    // EN: Fallback after override release.
    //     The discharge sequence should normally keep override active
    //     during return. If override is released unexpectedly, return to
    //     programmed position automatically.
    backstopLatchedTargetPositionMm := backstopProgrammedTargetPositionMm;
    backstopPositioningRequestActive := TRUE;

END_IF;


//==============================================================
// 5.2) Active target selection
//==============================================================
// EN: Discharge override has priority even if normal automatic mode is off.
//     Without override or positioning request, target remains latched,
//     but the axis does not move.
// PT: Override de descarte tem prioridade mesmo com o automático normal desligado.
IF systemRunEnable AND backstopTargetOverrideActive THEN

    backstopTargetPositionMm :=
        LIMIT(
            machineConfig.backstopMinPositionMm,
            backstopTargetOverridePositionMm,
            machineConfig.backstopMaxPositionMm
        );

ELSE

    backstopTargetPositionMm :=
        LIMIT(
            machineConfig.backstopMinPositionMm,
            backstopLatchedTargetPositionMm,
            machineConfig.backstopMaxPositionMm
        );

END_IF;


//==============================================================
// 5.4) Home running flag
//==============================================================
IF (backstopControlState = 10) OR
   (backstopControlState = 11) OR
   (backstopControlState = 12) OR
   (backstopControlState = 13) OR
   (backstopControlState = 14) THEN

    backstopHomeRunning := TRUE;

ELSE

    backstopHomeRunning := FALSE;

END_IF;


//==============================================================
// 6) Position error calculation
//==============================================================
backstopPositionErrorMm :=
    backstopTargetPositionMm - backstopPositionMm;

backstopAbsPositionErrorMm :=
    ABS(backstopPositionErrorMm);

backstopInPosition :=
    backstopHomed AND
    (backstopAbsPositionErrorMm <= machineConfig.backstopPositionToleranceMm);


//==============================================================
// 7) Reset fault command
//==============================================================
IF resetCmd THEN

    IF safetyCircuitOk AND
       backstopDriveOk AND
       NOT backstopSafeMaxLimit AND
       NOT backstopSafeMinLimit THEN

        backstopFault := FALSE;
        backstopFaultCode := 0;

        IF backstopControlState = 40 THEN
            backstopControlState := 0;
        END_IF

    END_IF

END_IF;


//==============================================================
// 8) General protection
//==============================================================
IF NOT safetyCircuitOk THEN

    backstopState := 'SAFETY_OFF';

    tonBackstopHomingTimeout(IN := FALSE);
    tonBackstopHomeSettleDelay(IN := FALSE);

    backstopFault := TRUE;
    backstopFaultCode := 2;
    backstopControlState := 40;


ELSIF NOT backstopDriveOk THEN

    backstopState := 'DRIVE_NOT_OK';

    tonBackstopHomingTimeout(IN := FALSE);
    tonBackstopHomeSettleDelay(IN := FALSE);

    backstopFault := TRUE;
    backstopFaultCode := 1;
    backstopControlState := 40;


ELSIF backstopSafeMaxLimit THEN

    backstopState := 'SAFE_MAX_LIMIT';

    tonBackstopHomingTimeout(IN := FALSE);
    tonBackstopHomeSettleDelay(IN := FALSE);

    backstopFault := TRUE;
    backstopFaultCode := 6;
    backstopControlState := 40;


ELSIF backstopSafeMinLimit THEN

    backstopState := 'SAFE_MIN_LIMIT';

    tonBackstopHomingTimeout(IN := FALSE);
    tonBackstopHomeSettleDelay(IN := FALSE);

    backstopFault := TRUE;
    backstopFaultCode := 7;
    backstopControlState := 40;


ELSIF machineConfig.backstopHomeDirection = 0 THEN

    backstopState := 'INVALID_HOME_DIR';

    tonBackstopHomingTimeout(IN := FALSE);
    tonBackstopHomeSettleDelay(IN := FALSE);

    backstopFault := TRUE;
    backstopFaultCode := 5;
    backstopControlState := 40;


ELSIF NOT systemRunEnable THEN

    // EN: Master stop disables movement without generating an axis fault.
    backstopState := 'SYSTEM_DISABLED';

    backstopSignedSpeedRefMmps := 0.0;

    tonBackstopHomingTimeout(IN := FALSE);
    tonBackstopHomeSettleDelay(IN := FALSE);

    backstopPositioningRequestActive := FALSE;

    IF backstopControlState <> 40 THEN
        backstopControlState := 0;
    END_IF


ELSE

    //==============================================================
    // 9) Mode selection
    //==============================================================
    // EN: Homing has priority over manual and automatic positioning.
    IF rBackstopHome AND NOT backstopFault THEN
        backstopControlState := 10;
    END_IF;


    //==============================================================
    // 10) Backstop state machine
    //==============================================================
    CASE backstopControlState OF

        0: // STOP
            backstopState := 'STOP';

            tonBackstopHomingTimeout(IN := FALSE);
            tonBackstopHomeSettleDelay(IN := FALSE);

            // EN: Manual is allowed even with auto enabled,
            //     but not during automatic cycle override.
            IF (backstopOpenCmd OR backstopCloseCmd) AND
               NOT backstopTargetOverrideActive THEN

                backstopControlState := 20;


            ELSIF backstopTargetOverrideActive OR
                  (
                      backstopAutoCmd AND
                      backstopPositioningRequestActive
                  ) THEN

                backstopControlState := 30;

            END_IF


        10: // HOME_FAST_SEARCH
            backstopState := 'HOME_FAST';

            backstopHomed := FALSE;
            backstopInPosition := FALSE;

            tonBackstopHomeSettleDelay(IN := FALSE);

            tonBackstopHomingTimeout(
                IN := TRUE,
                PT := machineConfig.backstopHomingTimeout
            );

            IF tonBackstopHomingTimeout.Q THEN

                backstopSignedSpeedRefMmps := 0.0;

                tonBackstopHomingTimeout(IN := FALSE);

                backstopFault := TRUE;
                backstopFaultCode := 3;

                backstopState := 'HOME_TIMEOUT';
                backstopControlState := 40;


            ELSIF backstopHomeLimitReached THEN

                backstopSignedSpeedRefMmps := 0.0;

                backstopControlState := 11;


            ELSE

                IF backstopHomeMoveAllowed THEN

                    IF machineConfig.backstopHomeDirection > 0 THEN

                        backstopSignedSpeedRefMmps :=
                            ABS(machineConfig.backstopHomingSpeedMmps);

                    ELSE

                        backstopSignedSpeedRefMmps :=
                            -ABS(machineConfig.backstopHomingSpeedMmps);

                    END_IF

                ELSE

                    backstopSignedSpeedRefMmps := 0.0;

                END_IF

            END_IF


        11: // HOME_SLOW_EXIT_SENSOR
            backstopState := 'HOME_SLOW_EXIT';

            tonBackstopHomeSettleDelay(IN := FALSE);

            tonBackstopHomingTimeout(
                IN := TRUE,
                PT := machineConfig.backstopHomingTimeout
            );

            IF tonBackstopHomingTimeout.Q THEN

                backstopSignedSpeedRefMmps := 0.0;

                tonBackstopHomingTimeout(IN := FALSE);

                backstopFault := TRUE;
                backstopFaultCode := 3;

                backstopState := 'HOME_TIMEOUT';
                backstopControlState := 40;


            ELSIF backstopHomeLimitFallingEdge THEN

                backstopSignedSpeedRefMmps := 0.0;

                tonBackstopHomingTimeout(IN := FALSE);

                backstopControlState := 12;


            ELSE

                IF backstopHomeMoveAllowed THEN

                    IF machineConfig.backstopHomeDirection > 0 THEN

                        backstopSignedSpeedRefMmps :=
                            -ABS(machineConfig.backstopMinMoveSpeedMmps);

                    ELSE

                        backstopSignedSpeedRefMmps :=
                            ABS(machineConfig.backstopMinMoveSpeedMmps);

                    END_IF

                ELSE

                    backstopSignedSpeedRefMmps := 0.0;

                END_IF

            END_IF


        12: // HOME_SET_ENCODER
            backstopState := 'HOME_SET_ENCODER';

            backstopSignedSpeedRefMmps := 0.0;

            tonBackstopHomingTimeout(IN := FALSE);
            tonBackstopHomeSettleDelay(IN := FALSE);

            // EN: Set encoder to configured known home position.
            backstopSetEncoderPositionTrigger := TRUE;
            backstopSetEncoderPositionMm := machineConfig.backstopHomePositionMm;

            backstopHomed := TRUE;
            backstopFault := FALSE;
            backstopFaultCode := 0;

            // EN: After homing, latch current programmed target for home move.
            backstopLatchedTargetPositionMm := backstopProgrammedTargetPositionMm;
            backstopPositioningRequestActive := TRUE;

            // EN: Homing cancels previous manual intervention memory.
            backstopManualInterventionActive := FALSE;
            backstopManualInterventionPositionMm := 0.0;

            backstopControlState := 13;


        13: // HOME_WAIT_AFTER_SET
            backstopState := 'HOME_WAIT';

            backstopSignedSpeedRefMmps := 0.0;

            tonBackstopHomingTimeout(IN := FALSE);

            // EN: Fixed wait after encoder set.
            tonBackstopHomeSettleDelay(
                IN := TRUE,
                PT := T#5S
            );

            IF tonBackstopHomeSettleDelay.Q THEN

                tonBackstopHomeSettleDelay(IN := FALSE);

                backstopControlState := 14;

            END_IF


        14: // HOME_MOVE_TO_TARGET
            backstopState := 'HOME_TO_TARGET';

            tonBackstopHomingTimeout(IN := FALSE);
            tonBackstopHomeSettleDelay(IN := FALSE);

            // EN: Move to the latched programmed target after homing.
            IF backstopInPosition THEN

                backstopSignedSpeedRefMmps := 0.0;

                backstopPositioningRequestActive := FALSE;

                // EN: Home positioning completed, no manual intervention pending.
                backstopManualInterventionActive := FALSE;
                backstopManualInterventionPositionMm := 0.0;

                backstopControlState := 0;


            ELSE

                backstopRawSpeedRefMmps :=
                    backstopPositionErrorMm * machineConfig.backstopPositionKp;

                backstopRawSpeedRefMmps :=
                    LIMIT(
                        -ABS(machineConfig.backstopAutoMaxSpeedMmps),
                        backstopRawSpeedRefMmps,
                        ABS(machineConfig.backstopAutoMaxSpeedMmps)
                    );

                IF ABS(backstopRawSpeedRefMmps) <
                   ABS(machineConfig.backstopMinMoveSpeedMmps) THEN

                    IF backstopPositionErrorMm > 0.0 THEN

                        backstopRawSpeedRefMmps :=
                            ABS(machineConfig.backstopMinMoveSpeedMmps);

                    ELSE

                        backstopRawSpeedRefMmps :=
                            -ABS(machineConfig.backstopMinMoveSpeedMmps);

                    END_IF

                END_IF

                IF (backstopRawSpeedRefMmps > 0.0) AND backstopOpenAllowed THEN

                    backstopSignedSpeedRefMmps := backstopRawSpeedRefMmps;

                ELSIF (backstopRawSpeedRefMmps < 0.0) AND backstopCloseAllowed THEN

                    backstopSignedSpeedRefMmps := backstopRawSpeedRefMmps;

                ELSE

                    backstopSignedSpeedRefMmps := 0.0;

                END_IF

            END_IF


        20: // MANUAL
            backstopState := 'MANUAL';

            tonBackstopHomingTimeout(IN := FALSE);
            tonBackstopHomeSettleDelay(IN := FALSE);

            // EN: If automatic override starts, manual is cancelled.
            IF backstopTargetOverrideActive THEN

                backstopSignedSpeedRefMmps := 0.0;
                backstopControlState := 30;


            ELSIF backstopOpenCmd AND backstopCloseCmd THEN

                backstopSignedSpeedRefMmps := 0.0;


            ELSIF backstopOpenCmd THEN

                IF backstopOpenAllowed THEN

                    backstopSignedSpeedRefMmps :=
                        ABS(machineConfig.backstopManualSpeedMmps);

                    // EN: Store last manual intervention position.
                    //     This is updated while the operator holds the manual command.
                    backstopManualInterventionActive := TRUE;
                    backstopManualInterventionPositionMm := backstopPositionMm;

                ELSE

                    backstopSignedSpeedRefMmps := 0.0;

                END_IF


            ELSIF backstopCloseCmd THEN

                IF backstopCloseAllowed THEN

                    backstopSignedSpeedRefMmps :=
                        -ABS(machineConfig.backstopManualSpeedMmps);

                    // EN: Store last manual intervention position.
                    //     Even if operator closes, the discharge sequence will use
                    //     MAX(programmed position, manual position), so it remains safe.
                    backstopManualInterventionActive := TRUE;
                    backstopManualInterventionPositionMm := backstopPositionMm;

                ELSE

                    backstopSignedSpeedRefMmps := 0.0;

                END_IF


            ELSE

                backstopSignedSpeedRefMmps := 0.0;

                // EN: After manual command release, do not automatically return
                //     to programmed position. Wait for execute positioning command.
                backstopPositioningRequestActive := FALSE;

                backstopControlState := 0;

            END_IF


        30: // AUTO_POSITION
            backstopState := 'AUTO_POSITION';

            tonBackstopHomingTimeout(IN := FALSE);
            tonBackstopHomeSettleDelay(IN := FALSE);

            IF NOT backstopAutoCmd AND
               NOT backstopTargetOverrideActive THEN

                backstopSignedSpeedRefMmps := 0.0;
                backstopPositioningRequestActive := FALSE;
                backstopControlState := 0;


            ELSIF NOT backstopHomed THEN

                backstopSignedSpeedRefMmps := 0.0;
                backstopState := 'AUTO_NO_HOME';


            ELSIF (backstopOpenCmd OR backstopCloseCmd) AND
                  NOT backstopTargetOverrideActive THEN

                // EN: Manual has priority only outside automatic cycle override.
                backstopSignedSpeedRefMmps := 0.0;
                backstopPositioningRequestActive := FALSE;
                backstopControlState := 20;


            ELSIF NOT backstopTargetOverrideActive AND
                  NOT backstopPositioningRequestActive THEN

                // EN: Auto enabled but no positioning command active.
                backstopSignedSpeedRefMmps := 0.0;
                backstopControlState := 0;


            ELSIF backstopInPosition THEN

                backstopSignedSpeedRefMmps := 0.0;

                // EN: Normal positioning command ends when target is reached.
                //     Override remains controlled by the automatic cycle.
                IF NOT backstopTargetOverrideActive THEN

                    backstopPositioningRequestActive := FALSE;

                    // EN: If the backstop returned to programmed target,
                    //     clear previous manual intervention memory.
                    backstopManualInterventionActive := FALSE;
                    backstopManualInterventionPositionMm := 0.0;

                    backstopControlState := 0;

                END_IF


            ELSE

                backstopRawSpeedRefMmps :=
                    backstopPositionErrorMm * machineConfig.backstopPositionKp;

                backstopRawSpeedRefMmps :=
                    LIMIT(
                        -ABS(machineConfig.backstopAutoMaxSpeedMmps),
                        backstopRawSpeedRefMmps,
                        ABS(machineConfig.backstopAutoMaxSpeedMmps)
                    );

                IF ABS(backstopRawSpeedRefMmps) <
                   ABS(machineConfig.backstopMinMoveSpeedMmps) THEN

                    IF backstopPositionErrorMm > 0.0 THEN

                        backstopRawSpeedRefMmps :=
                            ABS(machineConfig.backstopMinMoveSpeedMmps);

                    ELSE

                        backstopRawSpeedRefMmps :=
                            -ABS(machineConfig.backstopMinMoveSpeedMmps);

                    END_IF

                END_IF

                IF (backstopRawSpeedRefMmps > 0.0) AND backstopOpenAllowed THEN

                    backstopSignedSpeedRefMmps := backstopRawSpeedRefMmps;

                ELSIF (backstopRawSpeedRefMmps < 0.0) AND backstopCloseAllowed THEN

                    backstopSignedSpeedRefMmps := backstopRawSpeedRefMmps;

                ELSE

                    backstopSignedSpeedRefMmps := 0.0;

                END_IF

            END_IF


        40: // FAULT
            backstopState := 'FAULT';

            backstopSignedSpeedRefMmps := 0.0;

            tonBackstopHomingTimeout(IN := FALSE);
            tonBackstopHomeSettleDelay(IN := FALSE);

            backstopPositioningRequestActive := FALSE;

            IF resetCmd AND
               safetyCircuitOk AND
               backstopDriveOk AND
               NOT backstopSafeMaxLimit AND
               NOT backstopSafeMinLimit THEN

                backstopFault := FALSE;
                backstopFaultCode := 0;
                backstopControlState := 0;

            END_IF


    ELSE

        backstopControlState := 0;

    END_CASE;

END_IF;


//==============================================================
// 11) Encoder set pulse
//==============================================================
// EN: Extend encoder set command to ensure the encoder block sees it.
tpBackstopSetEncoderPosition(
    IN := backstopSetEncoderPositionTrigger,
    PT := machineConfig.backstopSetEncoderPulseTime
);

backstopSetEncoderPosition := tpBackstopSetEncoderPosition.Q;


//==============================================================
// 12) Backstop drive direction and speed outputs
//==============================================================
// EN: Convert signed internal speed command into direction outputs
//     and positive speed reference.
IF systemRunEnable AND
   safetyCircuitOk AND
   backstopDriveOk AND
   NOT backstopFault AND
   (ABS(backstopSignedSpeedRefMmps) >= machineConfig.backstopRunMinSpeedMmps) THEN

    // EN: The servo receives the signed speed reference directly.
    // PT: O servo recebe diretamente a referência de velocidade com sinal.
    backstopSpeedRefMmps := backstopSignedSpeedRefMmps;

    backstopRunFw :=
        backstopSignedSpeedRefMmps > 0.0;

    backstopRunRev :=
        backstopSignedSpeedRefMmps < 0.0;

ELSE

    backstopSpeedRefMmps := 0.0;

    backstopRunFw := FALSE;
    backstopRunRev := FALSE;

END_IF;

// EN: Enable the servo with the stacker system; drive-ready feedback is not used here
//     because it would create a circular enable dependency.
// PT: Habilita o servo com o sistema do stacker; o retorno de drive pronto não é usado
//     aqui porque criaria uma dependência circular de habilitação.
backstopDriveEnable := systemRunEnable AND safetyCircuitOk;


//==============================================================
// 13) Backstop plate lift solenoid
//==============================================================
// EN: Lift the backstop plate during backstop movement and homing.
//     Discharge conveyor protection can be ORed after all methods are called.
IF systemRunEnable AND
   (
       backstopRunFw OR
       backstopRunRev OR
       sheetStackDischargeConveyorRun OR
       (backstopControlState = 10) OR
       (backstopControlState = 11) OR
       (backstopControlState = 12) OR
       (backstopControlState = 13) OR
       (backstopControlState = 14)
   ) THEN

    backstopPlateUpSolenoid := TRUE;
    instTONBackstopDownDelay.IN := FALSE;

ELSE

    instTONBackstopDownDelay.IN := TRUE;

    IF instTONBackstopDownDelay.Q THEN

        backstopPlateUpSolenoid := FALSE;

    END_IF

END_IF;

instTONBackstopDownDelay(PT := T#200MS);
END_METHOD

//==============================================================
// COMPLEX STACKER — SPEED REFERENCE GENERATOR
// EN: Generates synchronized and sheet-stack separation speed references [m/min].
//==============================================================
METHOD _ConveyorSpeedControl
VAR
    rPackageComplete                  : BOOL;
    packageGapReady                   : BOOL;
    validCycleTimeS                   : REAL;

    sheetConveyorsSpeedUpReferenceMPM : REAL;

    sheetConveyor1BaseSpeedMPM        : REAL;
    sheetConveyor2BaseSpeedMPM        : REAL;
    sheetConveyor3BaseSpeedMPM        : REAL;
    sheetConveyor4BaseSpeedMPM        : REAL;
END_VAR


//==============================================================
// 1) Default event pulses
//==============================================================
sheetStackSeparationStarted         := FALSE;
sheetStackSeparationFinished        := FALSE;

sheetConveyor2SeparationStarted     := FALSE;
sheetConveyor2SeparationFinished    := FALSE;

sheetConveyor3SeparationStarted     := FALSE;
sheetConveyor3SeparationFinished    := FALSE;

sheetConveyor4SeparationStarted     := FALSE;
sheetConveyor4SeparationFinished    := FALSE;


//==============================================================
// 2) Edge detection
//==============================================================
rPackageComplete := packageCompleteCmd AND NOT packageCompleteCmdOld;
packageCompleteCmdOld := packageCompleteCmd;


//==============================================================
// 3) Enable and scan time
//==============================================================
speedControlEnabled :=
    sheetConveyor1Run AND
    sheetConveyor2Run AND
    sheetConveyor3Run AND
    sheetConveyor4Run AND
    safetyCircuitOk;

rampReset := NOT speedControlEnabled;


// EN: Read PLC scan time using OSCAT CYCLE_TIME.
instCycleTime(
    RST := resetCmd
);


// EN: Convert last cycle time from TIME/ms to seconds.
scanTimeMs := TIME_TO_REAL(instCycleTime.ct_last);

validCycleTimeS :=
    LIMIT(
        0.001,
        scanTimeMs / 1000.0,
        20.0
    );

scanTimeS := validCycleTimeS;


//==============================================================
// 4) Sheet length conversion
//==============================================================
// EN: Sheet length is kept converted for other calculations,
//     but it is no longer used as the separation tracking target.
sheetLengthM := MAX(0.0, sheetLengthMm) / 1000.0;


//==============================================================
// 5) Calculate normal stacker speed
//==============================================================
IF speedControlEnabled THEN

    normalStackerSpeedMPM :=
        LIMIT(
            machineConfig.minimumSpeedMPM,
            MAX(0.0, lineSpeedMPM) *
                MAX(0.0, machineConfig.stackerSpeedRatio),
            machineConfig.maximumSpeedMPM
        );

ELSE

    normalStackerSpeedMPM := 0.0;

END_IF;


//==============================================================
// 6) Calculate normal speed for each conveyor
//==============================================================
sheetConveyor1NormalSpeedMPM :=
    normalStackerSpeedMPM *
    MAX(0.0, machineConfig.sheetConveyor1SpeedTrim);

sheetConveyor2NormalSpeedMPM :=
    normalStackerSpeedMPM *
    MAX(0.0, machineConfig.sheetConveyor2SpeedTrim);

sheetConveyor3NormalSpeedMPM :=
    normalStackerSpeedMPM *
    MAX(0.0, machineConfig.sheetConveyor3SpeedTrim);

sheetConveyor4NormalSpeedMPM :=
    normalStackerSpeedMPM *
    MAX(0.0, machineConfig.sheetConveyor4SpeedTrim);


//==============================================================
// 6.1) Sheet conveyors speed-up reference
//==============================================================
// EN: Speed-up is added directly to conveyors 1/2/3 references.
//     It can work even when line speed is zero, as long as the
//     conveyor group is enabled.
IF speedControlEnabled AND sheetConveyorsSpeedUpCmd THEN

    sheetConveyorsSpeedUpReferenceMPM :=
        MAX(0.0, machineConfig.sheetConveyorsSpeedUpMPM);

ELSE

    sheetConveyorsSpeedUpReferenceMPM := 0.0;

END_IF;


//==============================================================
// 6.2) Base speed references including speed-up
//==============================================================
// EN: Base speed is the synchronized conveyor speed plus operator speed-up.
//     Separation tracking must use this base speed as reference.
sheetConveyor1BaseSpeedMPM :=
    sheetConveyor1NormalSpeedMPM + sheetConveyorsSpeedUpReferenceMPM;

sheetConveyor2BaseSpeedMPM :=
    sheetConveyor2NormalSpeedMPM + sheetConveyorsSpeedUpReferenceMPM;

sheetConveyor3BaseSpeedMPM :=
    sheetConveyor3NormalSpeedMPM + sheetConveyorsSpeedUpReferenceMPM;

sheetConveyor4BaseSpeedMPM :=
    sheetConveyor4NormalSpeedMPM + sheetConveyorsSpeedUpReferenceMPM;


//==============================================================
// 7) Calculate separation high speed
//==============================================================
// EN: Gap speed also receives the same speed-up reference.
//     This preserves the real gap differential while allowing operator boost.
sheetConveyor2GapSpeedMPM :=
    (sheetConveyor2NormalSpeedMPM * MAX(0.0, machineConfig.packageGapSpeedRatio)) +
    machineConfig.packageGapSpeedOffsetMPM +
    sheetConveyorsSpeedUpReferenceMPM;

sheetConveyor3GapSpeedMPM :=
    (sheetConveyor3NormalSpeedMPM * MAX(0.0, machineConfig.packageGapSpeedRatio)) +
    machineConfig.packageGapSpeedOffsetMPM +
    sheetConveyorsSpeedUpReferenceMPM;

sheetConveyor4GapSpeedMPM :=
    (sheetConveyor4NormalSpeedMPM * MAX(0.0, machineConfig.packageGapSpeedRatio)) +
    machineConfig.packageGapSpeedOffsetMPM +
    sheetConveyorsSpeedUpReferenceMPM;


//==============================================================
// 8) Calculate separation tracking target distances
//==============================================================
// EN: Separation tracking target is based on each conveyor length.
sheetConveyor2TargetDistanceM :=
    MAX(0.0, machineConfig.sheetConveyor2LengthM);

sheetConveyor3TargetDistanceM :=
    MAX(0.0, machineConfig.sheetConveyor3LengthM);

sheetConveyor4TargetDistanceM :=
    MAX(0.0, machineConfig.sheetConveyor4LengthM);


//==============================================================
// 9) Check separation ready conditions
//==============================================================
// EN: Compare gap speed against base speed, not normal speed.
//     Otherwise operator speed-up would be incorrectly counted as gap opening.
packageGapReady :=
    speedControlEnabled AND
    (sheetConveyor2TargetDistanceM > 0.0) AND
    (sheetConveyor3TargetDistanceM > 0.0) AND
    (sheetConveyor4TargetDistanceM > 0.0) AND
    ((sheetConveyor2GapSpeedMPM - sheetConveyor2BaseSpeedMPM) >= machineConfig.minimumOpeningSpeedMPM) AND
    ((sheetConveyor3GapSpeedMPM - sheetConveyor3BaseSpeedMPM) >= machineConfig.minimumOpeningSpeedMPM) AND
    ((sheetConveyor4GapSpeedMPM - sheetConveyor4BaseSpeedMPM) >= machineConfig.minimumOpeningSpeedMPM);

sheetStackSeparationReady := packageGapReady;


//==============================================================
// 10) Sheet stack separation state machine
//==============================================================
IF NOT speedControlEnabled THEN

    sheetStackSeparationState      := 'DISABLED';
    sheetStackSeparationStateCode  := -1;

    packageSeparationState         := 0;

    sheetStackSeparationActive     := FALSE;
    sheetStackBrakeActive          := FALSE;
    brakeValve                     := FALSE;

    sheetConveyor2SeparationActive := FALSE;
    sheetConveyor3SeparationActive := FALSE;
    sheetConveyor4SeparationActive := FALSE;

    sheetConveyor2HighSpeedActive  := FALSE;
    sheetConveyor3HighSpeedActive  := FALSE;
    sheetConveyor4HighSpeedActive  := FALSE;

    sheetConveyor2OpeningDistanceM := 0.0;
    sheetConveyor3OpeningDistanceM := 0.0;
    sheetConveyor4OpeningDistanceM := 0.0;

    sheetConveyor1TargetSpeedMPM   := 0.0;
    sheetConveyor2TargetSpeedMPM   := 0.0;
    sheetConveyor3TargetSpeedMPM   := 0.0;
    sheetConveyor4TargetSpeedMPM   := 0.0;


ELSE

    CASE packageSeparationState OF

        0: // NORMAL
            sheetStackSeparationState     := 'NORMAL';
            sheetStackSeparationStateCode := 0;

            sheetStackSeparationActive    := FALSE;
            sheetStackBrakeActive         := FALSE;
            brakeValve                    := FALSE;

            sheetConveyor2SeparationActive := FALSE;
            sheetConveyor3SeparationActive := FALSE;
            sheetConveyor4SeparationActive := FALSE;

            sheetConveyor2HighSpeedActive  := FALSE;
            sheetConveyor3HighSpeedActive  := FALSE;
            sheetConveyor4HighSpeedActive  := FALSE;

            sheetConveyor2OpeningDistanceM := 0.0;
            sheetConveyor3OpeningDistanceM := 0.0;
            sheetConveyor4OpeningDistanceM := 0.0;

            sheetConveyor1TargetSpeedMPM  := sheetConveyor1BaseSpeedMPM;
            sheetConveyor2TargetSpeedMPM  := sheetConveyor2BaseSpeedMPM;
            sheetConveyor3TargetSpeedMPM  := sheetConveyor3BaseSpeedMPM;
            sheetConveyor4TargetSpeedMPM  := sheetConveyor4BaseSpeedMPM;

            IF rPackageComplete AND packageGapReady THEN
                packageSeparationState := 10;
            END_IF


        10: // START_SHEET_STACK_SEPARATION
            sheetStackSeparationState     := 'START_SEPARATION';
            sheetStackSeparationStateCode := 10;

            sheetStackSeparationActive    := TRUE;
            sheetStackSeparationStarted   := TRUE;

            sheetStackBrakeActive         := TRUE;
            brakeValve                    := TRUE;

            // EN: Conveyor 2 tracking starts immediately.
            sheetConveyor2SeparationStarted := TRUE;

            sheetConveyor2SeparationActive  := TRUE;
            sheetConveyor3SeparationActive  := FALSE;
            sheetConveyor4SeparationActive  := FALSE;

            // EN: Conveyor 2 and 3 accelerate together from the beginning.
            sheetConveyor2HighSpeedActive   := TRUE;
            sheetConveyor3HighSpeedActive   := TRUE;
            sheetConveyor4HighSpeedActive   := TRUE;

            sheetConveyor2OpeningDistanceM  := 0.0;
            sheetConveyor3OpeningDistanceM  := 0.0;
            sheetConveyor4OpeningDistanceM  := 0.0;

            sheetConveyor1TargetSpeedMPM    := sheetConveyor1BaseSpeedMPM;
            sheetConveyor2TargetSpeedMPM    := sheetConveyor2GapSpeedMPM;
            sheetConveyor3TargetSpeedMPM    := sheetConveyor3GapSpeedMPM;
            sheetConveyor4TargetSpeedMPM    := sheetConveyor4GapSpeedMPM;

            packageSeparationState := 20;


        20: // SHEET_CONVEYOR_2_SEPARATION_TRACKING
            sheetStackSeparationState     := 'CONV2_TRACKING';
            sheetStackSeparationStateCode := 20;

            sheetStackSeparationActive    := TRUE;

            sheetStackBrakeActive         := TRUE;
            brakeValve                    := TRUE;

            sheetConveyor2SeparationActive := TRUE;
            sheetConveyor3SeparationActive := FALSE;
            sheetConveyor4SeparationActive := FALSE;

            sheetConveyor2HighSpeedActive  := TRUE;
            sheetConveyor3HighSpeedActive  := TRUE;
            sheetConveyor4HighSpeedActive  := TRUE;

            sheetConveyor1TargetSpeedMPM  := sheetConveyor1BaseSpeedMPM;
            sheetConveyor2TargetSpeedMPM  := sheetConveyor2GapSpeedMPM;
            sheetConveyor3TargetSpeedMPM  := sheetConveyor3GapSpeedMPM;
            sheetConveyor4TargetSpeedMPM  := sheetConveyor4GapSpeedMPM;

            IF sheetConveyor2OpeningDistanceM >= sheetConveyor2TargetDistanceM THEN

                // EN: Conveyor 2 tracking finished. Conveyor 2 returns to base speed.
                sheetConveyor2SeparationFinished := TRUE;

                sheetConveyor2SeparationActive   := FALSE;
                sheetConveyor2HighSpeedActive    := FALSE;

                sheetStackBrakeActive            := FALSE;
                brakeValve                       := FALSE;

                sheetConveyor2TargetSpeedMPM     := sheetConveyor2BaseSpeedMPM;

                // EN: Conveyor 3 tracking starts after conveyor 2 returns to sync.
                sheetConveyor3SeparationStarted := TRUE;
                sheetConveyor3OpeningDistanceM  := 0.0;

                packageSeparationState := 30;

            END_IF


        30: // SHEET_CONVEYOR_3_SEPARATION_TRACKING
            sheetStackSeparationState     := 'CONV3_TRACKING';
            sheetStackSeparationStateCode := 30;

            sheetStackSeparationActive    := TRUE;

            sheetStackBrakeActive         := FALSE;
            brakeValve                    := FALSE;

            sheetConveyor2SeparationActive := FALSE;
            sheetConveyor3SeparationActive := TRUE;
            sheetConveyor4SeparationActive := FALSE;

            sheetConveyor2HighSpeedActive  := FALSE;
            sheetConveyor3HighSpeedActive  := TRUE;
            sheetConveyor4HighSpeedActive  := TRUE;

            sheetConveyor1TargetSpeedMPM  := sheetConveyor1BaseSpeedMPM;
            sheetConveyor2TargetSpeedMPM  := sheetConveyor2BaseSpeedMPM;
            sheetConveyor3TargetSpeedMPM  := sheetConveyor3GapSpeedMPM;
            sheetConveyor4TargetSpeedMPM  := sheetConveyor4GapSpeedMPM;

            IF sheetConveyor3OpeningDistanceM >= sheetConveyor3TargetDistanceM THEN

                // EN: Conveyor 3 returns to base synchronized speed.
                sheetConveyor3TargetSpeedMPM := sheetConveyor3BaseSpeedMPM;

                // EN: Conveyor 4 tracking starts after conveyor 3 returns to sync.
                // PT: O rastreamento da esteira 4 inicia após a esteira 3 retornar ao sincronismo.
                sheetConveyor4SeparationStarted := TRUE;
                sheetConveyor4OpeningDistanceM := 0.0;

                packageSeparationState := 40;

            END_IF


        40: // SHEET_CONVEYOR_4_SEPARATION_TRACKING
            sheetStackSeparationState     := 'CONV4_TRACKING';
            sheetStackSeparationStateCode := 40;

            sheetStackSeparationActive    := TRUE;
            sheetStackBrakeActive         := FALSE;
            brakeValve                    := FALSE;

            sheetConveyor2SeparationActive := FALSE;
            sheetConveyor3SeparationActive := FALSE;
            sheetConveyor4SeparationActive := TRUE;

            sheetConveyor2HighSpeedActive := FALSE;
            sheetConveyor3HighSpeedActive := FALSE;
            sheetConveyor4HighSpeedActive := TRUE;

            sheetConveyor1TargetSpeedMPM := sheetConveyor1BaseSpeedMPM;
            sheetConveyor2TargetSpeedMPM := sheetConveyor2BaseSpeedMPM;
            sheetConveyor3TargetSpeedMPM := sheetConveyor3BaseSpeedMPM;
            sheetConveyor4TargetSpeedMPM := sheetConveyor4GapSpeedMPM;

            IF sheetConveyor4OpeningDistanceM >= sheetConveyor4TargetDistanceM THEN
                sheetConveyor4TargetSpeedMPM := sheetConveyor4BaseSpeedMPM;
                packageSeparationState := 50;
            END_IF


        50: // FINISH_SHEET_STACK_SEPARATION
            sheetStackSeparationState     := 'FINISH_SEPARATION';
            sheetStackSeparationStateCode := 50;

            sheetStackSeparationActive    := FALSE;
            sheetStackSeparationFinished  := TRUE;

            sheetStackBrakeActive         := FALSE;
            brakeValve                    := FALSE;

            sheetConveyor2SeparationActive  := FALSE;
            sheetConveyor3SeparationActive  := FALSE;
            sheetConveyor4SeparationActive  := FALSE;

            sheetConveyor2HighSpeedActive   := FALSE;
            sheetConveyor3HighSpeedActive   := FALSE;
            sheetConveyor4HighSpeedActive   := FALSE;

            sheetConveyor3SeparationFinished := TRUE;
            sheetConveyor4SeparationFinished := TRUE;

            sheetConveyor1TargetSpeedMPM  := sheetConveyor1BaseSpeedMPM;
            sheetConveyor2TargetSpeedMPM  := sheetConveyor2BaseSpeedMPM;
            sheetConveyor3TargetSpeedMPM  := sheetConveyor3BaseSpeedMPM;
            sheetConveyor4TargetSpeedMPM  := sheetConveyor4BaseSpeedMPM;

            packageSeparationState := 0;


    ELSE

        packageSeparationState := 0;

    END_CASE;

END_IF;


//==============================================================
// 11) Limit speed targets
//==============================================================
sheetConveyor1TargetSpeedMPM := LIMIT(
    machineConfig.minimumSpeedMPM,
    sheetConveyor1TargetSpeedMPM,
    machineConfig.maximumSpeedMPM
);

sheetConveyor2TargetSpeedMPM := LIMIT(
    machineConfig.minimumSpeedMPM,
    sheetConveyor2TargetSpeedMPM,
    machineConfig.maximumSpeedMPM
);

sheetConveyor3TargetSpeedMPM := LIMIT(
    machineConfig.minimumSpeedMPM,
    sheetConveyor3TargetSpeedMPM,
    machineConfig.maximumSpeedMPM
);

sheetConveyor4TargetSpeedMPM := LIMIT(
    machineConfig.minimumSpeedMPM,
    sheetConveyor4TargetSpeedMPM,
    machineConfig.maximumSpeedMPM
);


//==============================================================
// 12) Ramp sheet conveyor 1 speed reference
//==============================================================
instRampSheetConveyor1(
    X          := sheetConveyor1TargetSpeedMPM,
    A_UP       := MAX(0.0, machineConfig.rampAccelerationUpMPMps2),
    A_DN       := -MAX(0.0, machineConfig.rampAccelerationDownMPMps2),
    VU_MAX     := MAX(0.0, machineConfig.rampVelocityUpMaxMPMps),
    VD_MAX     := -MAX(0.0, machineConfig.rampVelocityDownMaxMPMps),
    LIMIT_HIGH := machineConfig.maximumSpeedMPM,
    LIMIT_LOW  := machineConfig.minimumSpeedMPM,
    RST        := rampReset,
    Y          => sheetConveyor1SpeedRefMPM
);


//==============================================================
// 13) Ramp sheet conveyor 2 speed reference
//==============================================================
instRampSheetConveyor2(
    X          := sheetConveyor2TargetSpeedMPM,
    A_UP       := MAX(0.0, machineConfig.rampAccelerationUpMPMps2),
    A_DN       := -MAX(0.0, machineConfig.rampAccelerationDownMPMps2),
    VU_MAX     := MAX(0.0, machineConfig.rampVelocityUpMaxMPMps),
    VD_MAX     := -MAX(0.0, machineConfig.rampVelocityDownMaxMPMps),
    LIMIT_HIGH := machineConfig.maximumSpeedMPM,
    LIMIT_LOW  := machineConfig.minimumSpeedMPM,
    RST        := rampReset,
    Y          => sheetConveyor2SpeedRefMPM
);


//==============================================================
// 14) Ramp sheet conveyor 3 speed reference
//==============================================================
instRampSheetConveyor3(
    X          := sheetConveyor3TargetSpeedMPM,
    A_UP       := MAX(0.0, machineConfig.rampAccelerationUpMPMps2),
    A_DN       := -MAX(0.0, machineConfig.rampAccelerationDownMPMps2),
    VU_MAX     := MAX(0.0, machineConfig.rampVelocityUpMaxMPMps),
    VD_MAX     := -MAX(0.0, machineConfig.rampVelocityDownMaxMPMps),
    LIMIT_HIGH := machineConfig.maximumSpeedMPM,
    LIMIT_LOW  := machineConfig.minimumSpeedMPM,
    RST        := rampReset,
    Y          => sheetConveyor3SpeedRefMPM
);


//==============================================================
// 15) Ramp sheet conveyor 4 speed reference
//==============================================================
instRampSheetConveyor4(
    X          := sheetConveyor4TargetSpeedMPM,
    A_UP       := MAX(0.0, machineConfig.rampAccelerationUpMPMps2),
    A_DN       := -MAX(0.0, machineConfig.rampAccelerationDownMPMps2),
    VU_MAX     := MAX(0.0, machineConfig.rampVelocityUpMaxMPMps),
    VD_MAX     := -MAX(0.0, machineConfig.rampVelocityDownMaxMPMps),
    LIMIT_HIGH := machineConfig.maximumSpeedMPM,
    LIMIT_LOW  := machineConfig.minimumSpeedMPM,
    RST        := rampReset,
    Y          => sheetConveyor4SpeedRefMPM
);


//==============================================================
// 16) Calculate real separation tracking speed using ramped references
//==============================================================
// EN: Only the real speed differential above the base speed moves the
//     separation point through the conveyors.
//     Operator speed-up is already included in base speed, so it is not
//     counted as gap opening.
sheetConveyor2OpeningSpeedMPM :=
    MAX(0.0, sheetConveyor2SpeedRefMPM - sheetConveyor2BaseSpeedMPM);

sheetConveyor3OpeningSpeedMPM :=
    MAX(0.0, sheetConveyor3SpeedRefMPM - sheetConveyor3BaseSpeedMPM);

sheetConveyor4OpeningSpeedMPM :=
    MAX(0.0, sheetConveyor4SpeedRefMPM - sheetConveyor4BaseSpeedMPM);


//==============================================================
// 17) Integrate real separation tracking distance
//==============================================================
IF speedControlEnabled THEN

    IF packageSeparationState = 20 THEN

        IF sheetConveyor2OpeningSpeedMPM >= machineConfig.minimumOpeningSpeedMPM THEN

            sheetConveyor2OpeningDistanceM :=
                sheetConveyor2OpeningDistanceM +
                (sheetConveyor2OpeningSpeedMPM / 60.0) * scanTimeS;

        END_IF

    ELSIF packageSeparationState = 30 THEN

        IF sheetConveyor3OpeningSpeedMPM >= machineConfig.minimumOpeningSpeedMPM THEN

            sheetConveyor3OpeningDistanceM :=
                sheetConveyor3OpeningDistanceM +
                (sheetConveyor3OpeningSpeedMPM / 60.0) * scanTimeS;

        END_IF

    ELSIF packageSeparationState = 40 THEN

        IF sheetConveyor4OpeningSpeedMPM >= machineConfig.minimumOpeningSpeedMPM THEN

            sheetConveyor4OpeningDistanceM :=
                sheetConveyor4OpeningDistanceM +
                (sheetConveyor4OpeningSpeedMPM / 60.0) * scanTimeS;

        END_IF

    END_IF

END_IF;


//==============================================================
// 18) Publish tracking distances to outputs
//==============================================================
sheetConveyor2TrackingDistanceM := sheetConveyor2OpeningDistanceM;
sheetConveyor3TrackingDistanceM := sheetConveyor3OpeningDistanceM;
sheetConveyor4TrackingDistanceM := sheetConveyor4OpeningDistanceM;
END_METHOD

//==============================================================
// COMPLEX STACKER - ELEVATOR CONTROL
// EN: Controls homing, manual movement, automatic leveling,
//     discharge positioning and magnetic brake timing.
// PT: Controla homing, movimento manual, nivelamento automático,
//     posicionamento de descarga e temporização do freio magnético.
//
// Signed speed: positive = up; negative = down.
// Velocidade com sinal: positivo = subir; negativo = descer.
//
// State code:
// 0  = STOP
// 10 = HOME_DOWN_SEARCH
// 11 = HOME_RELEASE_SENSOR
// 12 = HOME_SETTLE
// 13 = HOME_SET_ENCODER
// 14 = HOME_MOVE_TO_UPPER_POSITION
// 20 = MANUAL
// 30 = AUTO_LEVELING
// 40 = DISCHARGE_POSITIONING
// 90 = FAULT
//==============================================================
METHOD _ElevatorControl
//==============================================================
// 1) Default internal commands
//==============================================================
elevatorSignedSpeedRefMmps := 0.0;
elevatorSetEncoderPositionTrigger := FALSE;
elevatorManualLowSpeedZoneActive := FALSE;


//==============================================================
// 2) Homing request and lower sensor edge detection
//==============================================================
elevatorHomeRequestCombined :=
    systemRunEnable AND
    (
        elevatorHomeCmd OR
        (
            elevatorAutoCmd AND
            elevatorAutoHomeRequest
        )
    );

rElevatorHome :=
    elevatorHomeRequestCombined AND
    NOT elevatorHomeRequestCombinedOld;

elevatorHomeRequestCombinedOld := elevatorHomeRequestCombined;

elevatorHomeLimitReached := elevatorLowerLimit;

elevatorHomeLimitFallingEdge :=
    elevatorHomeLimitOld AND
    NOT elevatorHomeLimitReached;

elevatorHomeLimitOld := elevatorHomeLimitReached;


//==============================================================
// 2.1) Manual command rearm
//==============================================================
// EN: Manual commands held during homing or discharge must be released
//     before a new manual movement can start.
// PT: Comandos manuais mantidos durante homing ou descarte devem ser
//     liberados antes que um novo movimento manual possa iniciar.
IF NOT systemRunEnable OR
   NOT safetyCircuitOk OR
   NOT elevatorDriveOk OR
   elevatorFault OR
   (
        (elevatorControlState >= 10) AND
        (elevatorControlState <= 14)
   ) OR
   (elevatorControlState = 40) OR
   (elevatorControlState = 90) OR
   elevatorTargetOverrideActive OR
   sheetStackDischargeActive OR
   sheetStackDischargePending THEN

    elevatorManualCommandArmed := FALSE;

ELSIF NOT elevatorUpCmd AND
      NOT elevatorDownCmd THEN

    elevatorManualCommandArmed := TRUE;

END_IF;

elevatorManualCommandRequest :=
    elevatorManualCommandArmed AND
    (elevatorUpCmd OR elevatorDownCmd);


//==============================================================
// 3) Movement permissions
//==============================================================
elevatorUpAllowed :=
    systemRunEnable AND
    safetyCircuitOk AND
    elevatorDriveOk AND
    NOT elevatorUpperLimit AND
    NOT elevatorUpperSafetyLimit AND
    NOT backstopMaterialInterlockSensor AND
    (
        (NOT elevatorHomed) OR
        (elevatorPositionMm < machineConfig.elevatorMaxPositionMm)
    );

elevatorDownAllowed :=
    systemRunEnable AND
    safetyCircuitOk AND
    elevatorDriveOk AND
    NOT elevatorLowerLimit AND
    NOT elevatorLowerSafetyLimit AND
    (
        (NOT elevatorHomed) OR
        (elevatorPositionMm > machineConfig.elevatorMinPositionMm)
    );

// EN: Homing search ignores the normal lower limit until it is detected.
// PT: A busca de home ignora o limite inferior normal até detectá-lo.
elevatorHomeDownAllowed :=
    systemRunEnable AND
    safetyCircuitOk AND
    elevatorDriveOk AND
    NOT elevatorLowerSafetyLimit;

// EN: Upward release respects the backstop material interlock.
// PT: A liberação para cima respeita o intertravamento de material do backstop.
elevatorHomeReleaseAllowed :=
    systemRunEnable AND
    safetyCircuitOk AND
    elevatorDriveOk AND
    NOT elevatorUpperLimit AND
    NOT elevatorUpperSafetyLimit AND
    NOT backstopMaterialInterlockSensor;

//==============================================================
// 4) Target and position feedback
//==============================================================
IF elevatorControlState = 14 THEN

    elevatorTargetPositionMm := machineConfig.elevatorMaxPositionMm;

ELSIF elevatorTargetOverrideActive THEN

    elevatorTargetPositionMm :=
        LIMIT(
            machineConfig.elevatorMinPositionMm,
            elevatorTargetOverridePositionMm,
            machineConfig.elevatorMaxPositionMm
        );

ELSE

    elevatorTargetPositionMm :=
        LIMIT(
            machineConfig.elevatorMinPositionMm,
            elevatorPositionMm,
            machineConfig.elevatorMaxPositionMm
        );

END_IF;

elevatorPositionErrorMm :=
    elevatorTargetPositionMm - elevatorPositionMm;

elevatorAbsPositionErrorMm := ABS(elevatorPositionErrorMm);

// EN: Proportional position control with independent directional limits.
//     No minimum speed is forced; the servo may receive zero near the target.
// PT: Controle proporcional de posição com limites independentes por sentido.
//     Não força velocidade mínima; o servo pode receber zero próximo ao alvo.
elevatorRawSpeedRefMmps :=
    elevatorPositionErrorMm * MAX(0.0, machineConfig.elevatorPositionKp);

elevatorRawSpeedRefMmps :=
    LIMIT(
        -ABS(machineConfig.elevatorAutomaticDownSpeedMmps),
        elevatorRawSpeedRefMmps,
        ABS(machineConfig.elevatorAutomaticUpSpeedMmps)
    );

// EN: Endpoint flags depend on actual feedback and remain valid
//     independently of the active automatic target.
// PT: As flags de extremidade dependem do feedback real e permanecem
//     válidas independentemente do alvo automático ativo.
elevatorAtMinPosition :=
    elevatorHomed AND
    (
        elevatorLowerLimit OR
        (
            elevatorPositionMm <=
            (
                machineConfig.elevatorMinPositionMm +
                MAX(0.0, machineConfig.elevatorPositionToleranceMm)
            )
        )
    );

elevatorAtMaxPosition :=
    elevatorHomed AND
    (
        elevatorUpperLimit OR
        (
            elevatorPositionMm >=
            (
                machineConfig.elevatorMaxPositionMm -
                MAX(0.0, machineConfig.elevatorPositionToleranceMm)
            )
        )
    );

elevatorInPosition :=
    elevatorHomed AND
    (
        (elevatorAbsPositionErrorMm <= machineConfig.elevatorPositionToleranceMm)
        OR
        (
            elevatorUpperLimit AND
            (elevatorTargetPositionMm >= machineConfig.elevatorMaxPositionMm)
        )
        OR
        (
            elevatorLowerLimit AND
            (elevatorTargetPositionMm <= machineConfig.elevatorMinPositionMm)
        )
    );


//==============================================================
// 5) Fault reset
//==============================================================
IF resetCmd AND
   safetyCircuitOk AND
   elevatorDriveOk AND
   NOT elevatorUpperSafetyLimit AND
   NOT elevatorLowerSafetyLimit THEN

    elevatorFault := FALSE;
    elevatorFaultCode := 0;

    IF elevatorControlState = 90 THEN
        elevatorControlState := 0;
    END_IF

END_IF;


//==============================================================
// 6) Invalidate an interrupted homing sequence
//==============================================================
// EN: If homing or its final upward movement is interrupted by a
//     protection/system stop, a new homing cycle is required.
// PT: Se o homing ou sua subida final for interrompido por proteção/parada,
//     um novo ciclo de homing será obrigatório.
IF (elevatorControlState >= 10) AND
   (elevatorControlState <= 14) AND
   (
       NOT systemRunEnable OR
       NOT safetyCircuitOk OR
       NOT elevatorDriveOk OR
       elevatorUpperSafetyLimit OR
       elevatorLowerSafetyLimit
   ) THEN

    elevatorHomed := FALSE;
    elevatorReadyForAutomaticCycle := FALSE;

END_IF;


//==============================================================
// 7) General protection
//==============================================================
IF NOT safetyCircuitOk THEN

    elevatorState := 'SAFETY_OFF';
    elevatorFault := TRUE;
    elevatorFaultCode := 2;
    elevatorControlState := 90;

    tonElevatorHomingTimeout(IN := FALSE);
    tonElevatorHomeSettleDelay(IN := FALSE);
    tonElevatorLevelingSpeed2Delay(IN := FALSE);


ELSIF NOT elevatorDriveOk THEN

    elevatorState := 'DRIVE_NOT_OK';
    elevatorFault := TRUE;
    elevatorFaultCode := 1;
    elevatorControlState := 90;

    tonElevatorHomingTimeout(IN := FALSE);
    tonElevatorHomeSettleDelay(IN := FALSE);
    tonElevatorLevelingSpeed2Delay(IN := FALSE);


ELSIF elevatorUpperSafetyLimit THEN

    elevatorState := 'UPPER_SAFE_LIMIT';
    elevatorFault := TRUE;
    elevatorFaultCode := 4;
    elevatorControlState := 90;

    tonElevatorHomingTimeout(IN := FALSE);
    tonElevatorHomeSettleDelay(IN := FALSE);
    tonElevatorLevelingSpeed2Delay(IN := FALSE);


ELSIF elevatorLowerSafetyLimit THEN

    elevatorState := 'LOWER_SAFE_LIMIT';
    elevatorFault := TRUE;
    elevatorFaultCode := 5;
    elevatorControlState := 90;

    tonElevatorHomingTimeout(IN := FALSE);
    tonElevatorHomeSettleDelay(IN := FALSE);
    tonElevatorLevelingSpeed2Delay(IN := FALSE);


ELSIF NOT systemRunEnable THEN

    elevatorState := 'SYSTEM_DISABLED';
    elevatorSignedSpeedRefMmps := 0.0;

    tonElevatorHomingTimeout(IN := FALSE);
    tonElevatorHomeSettleDelay(IN := FALSE);
    tonElevatorLevelingSpeed2Delay(IN := FALSE);

    IF elevatorControlState <> 90 THEN
        elevatorControlState := 0;
    END_IF


ELSE

    //==========================================================
    // 8) Mode selection
    //==========================================================
    // EN: A new home command is ignored while discharge is active/pending.
    // PT: Novo comando de home é ignorado durante descarte ativo/pendente.
    IF rElevatorHome AND
       NOT elevatorFault AND
       NOT sheetStackDischargeActive AND
       NOT sheetStackDischargePending THEN

        elevatorControlState := 10;

    END_IF;

    // EN: Discharge override blocks manual and leveling commands.
    // PT: Override de descarte bloqueia comandos manuais e nivelamento.
    IF elevatorTargetOverrideActive AND
       elevatorHomed AND
       (elevatorControlState <> 10) AND
       (elevatorControlState <> 11) AND
       (elevatorControlState <> 12) AND
       (elevatorControlState <> 13) AND
       (elevatorControlState <> 14) AND
       (elevatorControlState <> 90) THEN

        elevatorControlState := 40;

    END_IF;


    //==========================================================
    // 9) Elevator state machine
    //==========================================================
    CASE elevatorControlState OF

        0: // STOP
            elevatorState := 'STOP';

            tonElevatorHomingTimeout(IN := FALSE);
            tonElevatorHomeSettleDelay(IN := FALSE);
            tonElevatorLevelingSpeed2Delay(IN := FALSE);

            // EN: Manual movement is available with automatic mode off.
            //     With automatic mode on, it is available only after homing
            //     and completion of the upper home positioning.
            // PT: O movimento manual fica disponível com o automático desligado.
            //     Com o automático ligado, fica disponível somente após o homing
            //     e a conclusão do posicionamento superior.
            IF elevatorManualCommandRequest AND
               (
                   NOT elevatorAutoCmd OR
                   (
                       elevatorHomed AND
                       elevatorReadyForAutomaticCycle
                   )
               ) THEN

                elevatorControlState := 20;

            ELSIF elevatorAutoCmd AND
                  elevatorHomed AND
                  elevatorReadyForAutomaticCycle THEN

                elevatorControlState := 30;

            END_IF


        10: // HOME_DOWN_SEARCH
            elevatorState := 'HOME_DOWN';
            elevatorHomed := FALSE;
            elevatorReadyForAutomaticCycle := FALSE;
            elevatorInPosition := FALSE;

            tonElevatorHomingTimeout(
                IN := TRUE,
                PT := machineConfig.elevatorHomingTimeout
            );

            IF tonElevatorHomingTimeout.Q THEN

                elevatorSignedSpeedRefMmps := 0.0;
                tonElevatorHomingTimeout(IN := FALSE);

                elevatorFault := TRUE;
                elevatorFaultCode := 3;
                elevatorState := 'HOME_TIMEOUT';
                elevatorControlState := 90;

            ELSIF elevatorHomeLimitReached THEN

                elevatorSignedSpeedRefMmps := 0.0;
                tonElevatorHomingTimeout(IN := FALSE);
                elevatorControlState := 11;

            ELSIF elevatorHomeDownAllowed THEN

                elevatorSignedSpeedRefMmps :=
                    -ABS(machineConfig.elevatorHomingSpeedMmps);

            END_IF


        11: // HOME_RELEASE_SENSOR
            elevatorState := 'HOME_RELEASE';

            tonElevatorHomingTimeout(
                IN := TRUE,
                PT := machineConfig.elevatorHomingTimeout
            );

            IF tonElevatorHomingTimeout.Q THEN

                elevatorSignedSpeedRefMmps := 0.0;
                tonElevatorHomingTimeout(IN := FALSE);

                elevatorFault := TRUE;
                elevatorFaultCode := 3;
                elevatorState := 'HOME_TIMEOUT';
                elevatorControlState := 90;

            ELSIF elevatorHomeLimitFallingEdge THEN

                elevatorSignedSpeedRefMmps := 0.0;
                tonElevatorHomingTimeout(IN := FALSE);
                tonElevatorHomeSettleDelay(IN := FALSE);
                elevatorControlState := 12;

            ELSIF elevatorHomeReleaseAllowed THEN

                elevatorSignedSpeedRefMmps :=
                    ABS(machineConfig.elevatorHomingReleaseSpeedMmps);

            END_IF


        12: // HOME_SETTLE
            elevatorState := 'HOME_SETTLE';
            elevatorSignedSpeedRefMmps := 0.0;

            // EN: Encoder reset is allowed only while the lower sensor
            //     remains released throughout the settle time.
            // PT: Reset do encoder é permitido somente se o sensor inferior
            //     permanecer livre durante todo o tempo de estabilização.
            IF elevatorHomeLimitReached THEN

                tonElevatorHomeSettleDelay(IN := FALSE);
                elevatorControlState := 11;

            ELSE

                tonElevatorHomeSettleDelay(
                    IN := TRUE,
                    PT := machineConfig.elevatorHomeSettleDelay
                );

                IF tonElevatorHomeSettleDelay.Q THEN
                    tonElevatorHomeSettleDelay(IN := FALSE);
                    elevatorControlState := 13;
                END_IF

            END_IF


        13: // HOME_SET_ENCODER
            elevatorState := 'HOME_SET_ENCODER';
            elevatorSignedSpeedRefMmps := 0.0;

            elevatorSetEncoderPositionTrigger := TRUE;
            elevatorSetEncoderPositionMm := machineConfig.elevatorHomePositionMm;

            elevatorHomed := TRUE;
            elevatorFault := FALSE;
            elevatorFaultCode := 0;

            tonElevatorHomingTimeout(IN := FALSE);
            elevatorControlState := 14;


        14: // HOME_MOVE_TO_UPPER_POSITION
            elevatorState := 'HOME_MOVE_UP';

            tonElevatorHomingTimeout(
                IN := TRUE,
                PT := machineConfig.elevatorHomingTimeout
            );

            IF elevatorInPosition THEN

                elevatorSignedSpeedRefMmps := 0.0;
                tonElevatorHomingTimeout(IN := FALSE);
                elevatorReadyForAutomaticCycle := TRUE;

                IF elevatorAutoCmd THEN
                    elevatorControlState := 30;
                ELSE
                    elevatorControlState := 0;
                END_IF

            ELSIF tonElevatorHomingTimeout.Q THEN

                elevatorSignedSpeedRefMmps := 0.0;
                tonElevatorHomingTimeout(IN := FALSE);

                elevatorHomed := FALSE;
                elevatorReadyForAutomaticCycle := FALSE;
                elevatorFault := TRUE;
                elevatorFaultCode := 3;
                elevatorState := 'HOME_UP_TIMEOUT';
                elevatorControlState := 90;

            ELSIF (elevatorRawSpeedRefMmps > 0.0) AND elevatorUpAllowed THEN

                elevatorSignedSpeedRefMmps :=
                    elevatorRawSpeedRefMmps;

            ELSIF (elevatorRawSpeedRefMmps < 0.0) AND elevatorDownAllowed THEN

                elevatorSignedSpeedRefMmps :=
                    elevatorRawSpeedRefMmps;

            END_IF


        20: // MANUAL
            elevatorState := 'MANUAL';

            tonElevatorHomingTimeout(IN := FALSE);
            tonElevatorHomeSettleDelay(IN := FALSE);
            tonElevatorLevelingSpeed2Delay(IN := FALSE);

            // EN: Discharge pending/active cancels manual operation.
            // PT: Descarte pendente/ativo cancela a operação manual.
            IF sheetStackDischargePending OR
               sheetStackDischargeActive OR
               elevatorTargetOverrideActive THEN

                elevatorSignedSpeedRefMmps := 0.0;

                IF elevatorAutoCmd AND
                   elevatorHomed AND
                   elevatorReadyForAutomaticCycle THEN

                    elevatorControlState := 30;

                ELSE

                    elevatorControlState := 0;

                END_IF


            ELSIF elevatorAutoCmd AND
                  (
                      NOT elevatorHomed OR
                      NOT elevatorReadyForAutomaticCycle
                  ) THEN

                elevatorSignedSpeedRefMmps := 0.0;
                elevatorState := 'AUTO_NO_HOME';
                elevatorControlState := 0;

            ELSIF elevatorUpCmd AND elevatorDownCmd THEN

                elevatorSignedSpeedRefMmps := 0.0;

            ELSIF elevatorUpCmd THEN

                IF elevatorUpAllowed THEN

                    // EN: Reduce manual upward speed only while approaching
                    //     the configured maximum position.
                    // PT: Reduz a velocidade manual de subida somente durante
                    //     a aproximação da posição máxima configurada.
                    elevatorManualLowSpeedZoneActive :=
                        elevatorHomed AND
                        (
                            LIMIT(
                                0.0,
                                machineConfig.elevatorManualLowSpeedFactor,
                                1.0
                            ) < 1.0
                        ) AND
                        (
                            elevatorPositionMm >=
                            (
                                machineConfig.elevatorMaxPositionMm -
                                MAX(
                                    0.0,
                                    machineConfig.elevatorManualLowSpeedZoneMm
                                )
                            )
                        );

                    IF elevatorManualLowSpeedZoneActive THEN

                        elevatorSignedSpeedRefMmps :=
                            ABS(machineConfig.elevatorManualSpeedMmps) *
                            LIMIT(
                                0.0,
                                machineConfig.elevatorManualLowSpeedFactor,
                                1.0
                            );

                    ELSE

                        elevatorSignedSpeedRefMmps :=
                            ABS(machineConfig.elevatorManualSpeedMmps);

                    END_IF

                ELSE
                    elevatorSignedSpeedRefMmps := 0.0;
                END_IF

            ELSIF elevatorDownCmd THEN

                IF elevatorDownAllowed THEN

                    // EN: Reduce manual downward speed only while approaching
                    //     the configured minimum position.
                    // PT: Reduz a velocidade manual de descida somente durante
                    //     a aproximação da posição mínima configurada.
                    elevatorManualLowSpeedZoneActive :=
                        elevatorHomed AND
                        (
                            LIMIT(
                                0.0,
                                machineConfig.elevatorManualLowSpeedFactor,
                                1.0
                            ) < 1.0
                        ) AND
                        (
                            elevatorPositionMm <=
                            (
                                machineConfig.elevatorMinPositionMm +
                                MAX(
                                    0.0,
                                    machineConfig.elevatorManualLowSpeedZoneMm
                                )
                            )
                        );

                    IF elevatorManualLowSpeedZoneActive THEN

                        elevatorSignedSpeedRefMmps :=
                            -ABS(machineConfig.elevatorManualSpeedMmps) *
                            LIMIT(
                                0.0,
                                machineConfig.elevatorManualLowSpeedFactor,
                                1.0
                            );

                    ELSE

                        elevatorSignedSpeedRefMmps :=
                            -ABS(machineConfig.elevatorManualSpeedMmps);

                    END_IF

                ELSE
                    elevatorSignedSpeedRefMmps := 0.0;
                END_IF

            ELSE

                elevatorSignedSpeedRefMmps := 0.0;

                // EN: When manual intervention ends, automatic leveling
                //     may immediately evaluate the current level sensor.
                // PT: Ao terminar a intervenção manual, o nivelamento
                //     automático pode avaliar imediatamente o sensor atual.
                IF elevatorAutoCmd AND
                   elevatorHomed AND
                   elevatorReadyForAutomaticCycle THEN

                    elevatorControlState := 30;

                ELSE

                    elevatorControlState := 0;

                END_IF

            END_IF


        30: // AUTO_LEVELING
            elevatorState := 'AUTO_LEVELING';

            tonElevatorHomingTimeout(IN := FALSE);
            tonElevatorHomeSettleDelay(IN := FALSE);

            IF NOT elevatorAutoCmd THEN

                elevatorSignedSpeedRefMmps := 0.0;
                tonElevatorLevelingSpeed2Delay(IN := FALSE);
                elevatorControlState := 0;

            ELSIF NOT elevatorHomed OR
                  NOT elevatorReadyForAutomaticCycle THEN

                elevatorSignedSpeedRefMmps := 0.0;
                tonElevatorLevelingSpeed2Delay(IN := FALSE);
                elevatorState := 'AUTO_NO_HOME';

            ELSIF (elevatorUpCmd OR elevatorDownCmd) AND
                  NOT elevatorManualCommandArmed THEN

                // EN: A command held from homing or discharge inhibits
                //     leveling but cannot start a manual movement.
                // PT: Um comando mantido desde o homing ou descarte bloqueia
                //     o nivelamento, mas não pode iniciar movimento manual.
                elevatorSignedSpeedRefMmps := 0.0;
                tonElevatorLevelingSpeed2Delay(IN := FALSE);

            ELSIF elevatorManualCommandRequest AND
                  NOT sheetStackDischargePending AND
                  NOT sheetStackDischargeActive THEN

                // EN: Manual commands have priority over the level sensor.
                //     The speed-2 delay restarts after manual intervention.
                // PT: Os comandos manuais têm prioridade sobre o sensor de nível.
                //     O atraso da velocidade 2 reinicia após a intervenção manual.
                elevatorSignedSpeedRefMmps := 0.0;
                tonElevatorLevelingSpeed2Delay(IN := FALSE);
                elevatorControlState := 20;

            ELSIF backstopStackLevelSensor AND
                  elevatorDownAllowed THEN

                tonElevatorLevelingSpeed2Delay(
                    IN := TRUE,
                    PT := machineConfig.elevatorLevelingSpeed2Delay
                );

                IF tonElevatorLevelingSpeed2Delay.Q THEN
                    elevatorSignedSpeedRefMmps :=
                        -ABS(machineConfig.elevatorLevelingSpeed2Mmps);
                ELSE
                    elevatorSignedSpeedRefMmps :=
                        -ABS(machineConfig.elevatorLevelingSpeed1Mmps);
                END_IF

            ELSE

                elevatorSignedSpeedRefMmps := 0.0;
                tonElevatorLevelingSpeed2Delay(IN := FALSE);

            END_IF


        40: // DISCHARGE_POSITIONING
            elevatorState := 'DISCHARGE_POSITION';

            tonElevatorLevelingSpeed2Delay(IN := FALSE);

            IF NOT elevatorTargetOverrideActive THEN

                elevatorSignedSpeedRefMmps := 0.0;

                IF elevatorAutoCmd AND
                   elevatorHomed AND
                   elevatorReadyForAutomaticCycle THEN

                    elevatorControlState := 30;

                ELSE

                    elevatorControlState := 0;

                END_IF

            ELSIF elevatorInPosition THEN

                elevatorSignedSpeedRefMmps := 0.0;

            ELSIF (elevatorRawSpeedRefMmps > 0.0) AND elevatorUpAllowed THEN

                elevatorSignedSpeedRefMmps :=
                    elevatorRawSpeedRefMmps;

            ELSIF (elevatorRawSpeedRefMmps < 0.0) AND elevatorDownAllowed THEN

                elevatorSignedSpeedRefMmps :=
                    elevatorRawSpeedRefMmps;

            END_IF


        90: // FAULT
            elevatorState := 'FAULT';
            elevatorSignedSpeedRefMmps := 0.0;

            tonElevatorHomingTimeout(IN := FALSE);
            tonElevatorHomeSettleDelay(IN := FALSE);
            tonElevatorLevelingSpeed2Delay(IN := FALSE);


        ELSE
            elevatorControlState := 0;

    END_CASE;

END_IF;


//==============================================================
// 10) Encoder set pulse
//==============================================================
tpElevatorSetEncoderPosition(
    IN := elevatorSetEncoderPositionTrigger,
    PT := machineConfig.elevatorSetEncoderPulseTime
);

elevatorSetEncoderPosition := tpElevatorSetEncoderPosition.Q;


//==============================================================
// 11) Servo enable and magnetic brake control
//==============================================================
// EN: Keep the servo enabled with zero speed, following the backstop concept.
//     Drive-ready feedback is not used to avoid a circular enable dependency.
// PT: Mantém o servo habilitado com velocidade zero, seguindo o backstop.
//     O retorno de drive pronto não é usado para evitar dependência circular.
elevatorDriveEnable := systemRunEnable AND safetyCircuitOk;

elevatorMoveRequest :=
    systemRunEnable AND
    safetyCircuitOk AND
    elevatorDriveOk AND
    NOT elevatorFault AND
    (ABS(elevatorSignedSpeedRefMmps) > 0.0);

IF elevatorMoveRequest THEN

    elevatorBrakeReleaseRequest := TRUE;
    tonElevatorBrakeHoldDelay(IN := FALSE);

ELSE

    IF elevatorBrakeRelease THEN

        tonElevatorBrakeHoldDelay(
            IN := TRUE,
            PT := machineConfig.elevatorBrakeHoldTime
        );

        elevatorBrakeReleaseRequest :=
            NOT tonElevatorBrakeHoldDelay.Q;

    ELSE

        tonElevatorBrakeHoldDelay(IN := FALSE);
        elevatorBrakeReleaseRequest := FALSE;

    END_IF

END_IF;

elevatorBrakeRelease :=
    systemRunEnable AND
    safetyCircuitOk AND
    elevatorDriveOk AND
    NOT elevatorFault AND
    elevatorBrakeReleaseRequest;

tonElevatorBrakeReleaseDelay(
    IN := elevatorMoveRequest AND elevatorBrakeRelease,
    PT := machineConfig.elevatorBrakeReleaseDelay
);


//==============================================================
// 12) Direction and speed outputs
//==============================================================
IF elevatorMoveRequest AND
   elevatorBrakeRelease AND
   tonElevatorBrakeReleaseDelay.Q THEN

    elevatorSpeedRefMmps := elevatorSignedSpeedRefMmps;
    elevatorRunUp := elevatorSignedSpeedRefMmps > 0.0;
    elevatorRunDown := elevatorSignedSpeedRefMmps < 0.0;

ELSE

    elevatorSpeedRefMmps := 0.0;
    elevatorRunUp := FALSE;
    elevatorRunDown := FALSE;

END_IF;
END_METHOD

METHOD _ExternalCommands : BOOL
VAR_INPUT
END_VAR
END_METHOD

//==============================================================
// COMPLEX STACKER — HMI STATUS
// EN: Maps internal status, outputs, positions and diagnostics
//     to the HMI status structure.
//==============================================================
METHOD _HmiStatus



//==============================================================
// 1) System general status
//==============================================================
hmiStatus.systemRunEnable :=
    systemRunEnable;

hmiStatus.safetyCircuitOk :=
    safetyCircuitOk;

hmiStatus.faultActive :=
    faultActive OR
    backstopFault OR
    elevatorFault OR
    sheetStackDischargeFault OR
    sheetStackDischargeConveyorFault;

hmiStatus.deviceState :=
    deviceState;


//==============================================================
// 2) Sheet conveyor group status
//==============================================================
hmiStatus.synchronizedConveyorsRunning :=
    synchronizedConveyorsRunning;

hmiStatus.sheetConveyor1Run :=
    sheetConveyor1Run;

hmiStatus.sheetConveyor2Run :=
    sheetConveyor2Run;

hmiStatus.sheetConveyor3Run :=
    sheetConveyor3Run;

hmiStatus.sheetConveyor4Run :=
    sheetConveyor4Run;

hmiStatus.sheetConveyor1SpeedRefMPM :=
    sheetConveyor1SpeedRefMPM;

hmiStatus.sheetConveyor2SpeedRefMPM :=
    sheetConveyor2SpeedRefMPM;

hmiStatus.sheetConveyor3SpeedRefMPM :=
    sheetConveyor3SpeedRefMPM;

hmiStatus.sheetConveyor4SpeedRefMPM :=
    sheetConveyor4SpeedRefMPM;

hmiStatus.syncConveyorsState :=
    syncConveyorsState;


//==============================================================
// 3) Sheet stack separation status
//==============================================================
hmiStatus.sheetStackSeparationReady :=
    sheetStackSeparationReady;

hmiStatus.sheetStackSeparationActive :=
    sheetStackSeparationActive;

hmiStatus.sheetStackBrakeActive :=
    sheetStackBrakeActive;


//==============================================================
// 4) Sheet stack discharge sequence status
//==============================================================
hmiStatus.sheetStackDischargeState :=
    sheetStackDischargeState;

hmiStatus.sheetStackDischargeStateCode :=
    sheetStackDischargeStateCode;

hmiStatus.sheetStackDischargePending :=
    sheetStackDischargePending;

hmiStatus.sheetStackDischargeActive :=
    sheetStackDischargeActive;

hmiStatus.sheetStackDischargeStarted :=
    sheetStackDischargeStarted;

hmiStatus.sheetStackDischargeFinished :=
    sheetStackDischargeFinished;

hmiStatus.sheetStackDischargeFault :=
    sheetStackDischargeFault;

hmiStatus.sheetStackDischargeFaultCode :=
    sheetStackDischargeFaultCode;

hmiStatus.sheetStackDischargeLastCycleOk :=
    sheetStackDischargeLastCycleOk;

hmiStatus.sheetStackDischargeLastResultCode :=
    sheetStackDischargeLastResultCode;

hmiStatus.sheetStackDischargeLastFaultStepCode :=
    sheetStackDischargeLastFaultStepCode;

hmiStatus.sheetStackDischargeLastFaultCode :=
    sheetStackDischargeLastFaultCode;


//==============================================================
// 5) Sheet stack discharge conveyor status
//==============================================================
hmiStatus.sheetStackDischargeConveyorState :=
    sheetStackDischargeConveyorState;

hmiStatus.sheetStackDischargeConveyorRun :=
    sheetStackDischargeConveyorRun;

hmiStatus.sheetStackDischargeConveyorSpeedRefMPM :=
    sheetStackDischargeConveyorSpeedRefMPM;

hmiStatus.sheetStackDischargeConveyorFault :=
    sheetStackDischargeConveyorFault;

hmiStatus.sheetStackDischargeConveyorFaultCode :=
    sheetStackDischargeConveyorFaultCode;


//==============================================================
// 6) Backstop status
//==============================================================
hmiStatus.backstopState :=
    backstopState;

hmiStatus.backstopHomed :=
    backstopHomed;

hmiStatus.backstopHomeRunning :=
    backstopHomeRunning;

hmiStatus.backstopInPosition :=
    backstopInPosition;

hmiStatus.backstopPositionMm :=
    backstopPositionMm;

hmiStatus.backstopTargetPositionMm :=
    backstopTargetPositionMm;

hmiStatus.backstopPositionErrorMm :=
    backstopPositionErrorMm;

hmiStatus.backstopRunFw :=
    backstopRunFw;

hmiStatus.backstopRunRev :=
    backstopRunRev;

hmiStatus.backstopSpeedRefMmps :=
    backstopSpeedRefMmps;

hmiStatus.backstopPlateUpSolenoid :=
    backstopPlateUpSolenoid;

hmiStatus.backstopSetEncoderPosition :=
    backstopSetEncoderPosition;

hmiStatus.backstopSetEncoderPositionMm :=
    backstopSetEncoderPositionMm;

hmiStatus.backstopManualInterventionActive :=
    backstopManualInterventionActive;

hmiStatus.backstopManualInterventionPositionMm :=
    backstopManualInterventionPositionMm;

hmiStatus.backstopFault :=
    backstopFault;

hmiStatus.backstopFaultCode :=
    backstopFaultCode;


//==============================================================
// 7) Elevator status
//==============================================================
hmiStatus.elevatorState :=
    elevatorState;

hmiStatus.elevatorHomed :=
    elevatorHomed;

hmiStatus.elevatorInPosition :=
    elevatorInPosition;

hmiStatus.elevatorPositionMm :=
    elevatorPositionMm;

hmiStatus.elevatorTargetPositionMm :=
    elevatorTargetPositionMm;

hmiStatus.elevatorPositionErrorMm :=
    elevatorPositionErrorMm;

hmiStatus.elevatorRunUp :=
    elevatorRunUp;

hmiStatus.elevatorRunDown :=
    elevatorRunDown;

hmiStatus.elevatorBrakeRelease :=
    elevatorBrakeRelease;

hmiStatus.elevatorSpeedRefMmps :=
    elevatorSpeedRefMmps;

hmiStatus.elevatorSetEncoderPosition :=
    elevatorSetEncoderPosition;

hmiStatus.elevatorSetEncoderPositionMm :=
    elevatorSetEncoderPositionMm;

hmiStatus.elevatorFault :=
    elevatorFault;

hmiStatus.elevatorFaultCode :=
    elevatorFaultCode;


//==============================================================
// 8) Process values
//==============================================================
hmiStatus.lineSpeedMPM :=
    lineSpeedMPM;

hmiStatus.sheetLengthMm :=
    sheetLengthMm;

hmiStatus.stackHeightMm :=
    stackHeightMm;


//==============================================================
// 9) Input / drive status mirror
//==============================================================
hmiStatus.sheetConveyor1DriveOk :=
    sheetConveyor1DriveOk;

hmiStatus.sheetConveyor2DriveOk :=
    sheetConveyor2DriveOk;

hmiStatus.sheetConveyor3DriveOk :=
    sheetConveyor3DriveOk;

hmiStatus.sheetConveyor4DriveOk :=
    sheetConveyor4DriveOk;

hmiStatus.backstopDriveOk :=
    backstopDriveOk;

hmiStatus.elevatorDriveOk :=
    elevatorDriveOk;

hmiStatus.sheetStackDischargeConveyorDriveOk :=
    sheetStackDischargeConveyorDriveOk;
END_METHOD

METHOD _MachineAuxilary
VAR_INPUT
END_VAR
(*



stopMachinePulse :=
    NOT safetyCircuitOk OR
    NOT sheetConveyor1DriveOk OR
    NOT sheetConveyor2DriveOk OR
    NOT sheetConveyor3DriveOk;
	NOT backstopDriveOk
	NOT elevatorDriveOk
*)
noCrushRollersUpDownValve := noCrushRollersDownCmd;

stackerRunning := systemRunEnable;


reset := resetCmd;
END_METHOD

//==============================================================
// COMPLEX STACKER — SHEET CONVEYOR GROUP CONTROL
// EN: Controls the synchronized sheet conveyor group.
//     Start/stop command latch is handled by _SystemControl().
//==============================================================
METHOD _SheetConveyorGroupControl

//==============================================================
// 1) Conditions
//==============================================================
// EN: Only synchronized sheet conveyor drives are considered here.
// PT: Apenas os inversores das esteiras sincronizadas são considerados aqui.
allSynchronizedDrivesOk :=
    sheetConveyor1DriveOk AND
    sheetConveyor2DriveOk AND
    sheetConveyor3DriveOk AND
    sheetConveyor4DriveOk;


// EN: Synchronized conveyor group fault.
// PT: Falha do grupo de esteiras sincronizadas.
anyFault :=
    NOT safetyCircuitOk OR
    NOT allSynchronizedDrivesOk;

faultActive := anyFault;


//==============================================================
// 2) State machine
//==============================================================
CASE syncConveyorsState OF

    0: // IDLE
        deviceState := 'IDLE';

        sheetConveyor1Run := FALSE;
        sheetConveyor2Run := FALSE;
        sheetConveyor3Run := FALSE;
        sheetConveyor4Run := FALSE;

        synchronizedConveyorsRunning := FALSE;

        // EN: The group starts only when the master system is enabled
        //     and no conveyor group fault is active.
        IF systemRunEnable AND NOT anyFault THEN

            syncConveyorsState := 1;

        ELSIF systemRunEnable AND anyFault THEN

            syncConveyorsState := 10;

        END_IF


    1: // RUN
        deviceState := 'RUN';

        // EN: Outputs are also directly conditioned by systemRunEnable
        //     to avoid one-scan movement after a stop command.
        sheetConveyor1Run :=
            systemRunEnable AND
            safetyCircuitOk AND
            sheetConveyor1DriveOk;

        sheetConveyor2Run :=
            systemRunEnable AND
            safetyCircuitOk AND
            sheetConveyor2DriveOk;

        sheetConveyor3Run :=
            systemRunEnable AND
            safetyCircuitOk AND
            sheetConveyor3DriveOk;

        sheetConveyor4Run :=
            systemRunEnable AND
            safetyCircuitOk AND
            sheetConveyor4DriveOk;

        synchronizedConveyorsRunning :=
            sheetConveyor1Run AND
            sheetConveyor2Run AND
            sheetConveyor3Run AND
            sheetConveyor4Run;

        IF anyFault THEN

            syncConveyorsState := 10;

        ELSIF NOT systemRunEnable THEN

            syncConveyorsState := 0;

        END_IF


    10: // FAULT
        deviceState := 'FAULT';

        sheetConveyor1Run := FALSE;
        sheetConveyor2Run := FALSE;
        sheetConveyor3Run := FALSE;
        sheetConveyor4Run := FALSE;

        synchronizedConveyorsRunning := FALSE;

        // EN: Fault state is released only by reset and with all faults cleared.
        //     If systemRunEnable is still TRUE after reset, the group can start
        //     again from IDLE on the next scan.
        IF resetCmd AND NOT anyFault THEN

            syncConveyorsState := 0;

        END_IF


ELSE

    syncConveyorsState := 0;

END_CASE;
END_METHOD

//==============================================================
// COMPLEX STACKER — SHEET STACK DISCHARGE CONTROL
// EN: Controls the sheet stack discharge sequence after the sheet
//     conveyor separation cycle is completed.
//
// State code
// 0  = IDLE
// 5  = WAIT_SEPARATION
// 10 = START_DISCHARGE_POSITIONING
// 20 = WAIT_DISCHARGE_POSITION
// 30 = RUN_DISCHARGE_CONVEYOR_AND_WAIT_CLEAR
// 40 = START_RETURN_POSITIONING
// 50 = WAIT_RETURN_POSITION
// 60 = FINISH
// 90 = FAULT_HOLD
//
// Last result code
// 0 = No cycle executed yet
// 1 = Last cycle completed successfully
// 2 = Last cycle completed with manual backstop skip
// 3 = Last cycle completed/aborted by timeout
// 4 = Last cycle aborted by fault
//
// Fault code
// 0  = No fault
// 1  = Safety circuit not OK
// 2  = Sheet conveyor drive not OK
// 3  = Discharge conveyor drive/control fault
// 4  = Backstop drive/control fault
// 5  = Elevator drive/control fault
// 6  = Stacker stopped during cycle
// 10 = Wait separation timeout
// 20 = Backstop positioning timeout
// 30 = Discharge conveyor did not start timeout
// 31 = Elevator platform clear timeout
// 50 = Backstop return timeout
//==============================================================
METHOD _SheetStackDischargeControl
VAR
    abortCycle : BOOL;
    backstopDischargeReady : BOOL;
    elevatorPlatformClear : BOOL;
END_VAR


//==============================================================
// 1) Default event pulses
//==============================================================
sheetStackDischargeStarted  := FALSE;
sheetStackDischargeFinished := FALSE;

// EN: An empty platform is accepted even when no stack was present
//     at the beginning of the discharge cycle.
// PT: Plataforma vazia é aceita mesmo quando não havia pilha
//     no início do ciclo de descarte.
elevatorPlatformClear :=
    NOT elevatorStackPresentAtDischargeStart OR
    (
        elevatorStackExitClearSensor AND
        NOT elevatorStackPresentSensor
    );


//==============================================================
// 2) Default internal requests / overrides
//==============================================================
// EN: The sequence does not write the physical discharge conveyor outputs.
//     It only generates an internal request to the conveyor control method.
sheetStackDischargeConveyorRunRequest := FALSE;

backstopTargetOverrideActive := FALSE;
backstopTargetOverridePositionMm := 0.0;

elevatorTargetOverrideActive := FALSE;
elevatorTargetOverridePositionMm := 0.0;


//==============================================================
// 3) Edge detection
//==============================================================
// EN: Separate edge detector to avoid interfering with conveyor speed control.
rPackageCompleteDischarge :=
    packageCompleteCmd AND NOT packageCompleteCmdOldDischarge;

packageCompleteCmdOldDischarge := packageCompleteCmd;


//==============================================================
// 4) Fault condition
//==============================================================
// EN: Elevator drive, homing and position feedback are required
//     for safe discharge sequence progress.
// PT: Drive, homing e posição do elevador são obrigatórios
//     para o avanço seguro da sequência de descarte.
sheetStackDischargeFaultCondition :=
    NOT safetyCircuitOk OR
    NOT sheetConveyor1DriveOk OR
    NOT sheetConveyor2DriveOk OR
    NOT sheetConveyor3DriveOk OR
    NOT sheetConveyor4DriveOk OR
    NOT sheetStackDischargeConveyorDriveOk OR
    sheetStackDischargeConveyorFault OR
    NOT backstopDriveOk OR
    NOT backstopHomed OR
    backstopFault OR
    NOT elevatorDriveOk OR
    NOT elevatorHomed OR
    NOT elevatorReadyForAutomaticCycle OR
    elevatorFault;


//==============================================================
// 5) Fault code priority
//==============================================================
IF NOT safetyCircuitOk THEN

    sheetStackDischargeFaultCode := 1;

ELSIF NOT sheetConveyor1DriveOk OR
      NOT sheetConveyor2DriveOk OR
      NOT sheetConveyor3DriveOk OR
      NOT sheetConveyor4DriveOk THEN

    sheetStackDischargeFaultCode := 2;

ELSIF NOT sheetStackDischargeConveyorDriveOk OR
      sheetStackDischargeConveyorFault THEN

    sheetStackDischargeFaultCode := 3;

ELSIF NOT backstopDriveOk OR
      NOT backstopHomed OR
      backstopFault THEN

    sheetStackDischargeFaultCode := 4;

ELSIF NOT elevatorDriveOk OR
      NOT elevatorHomed OR
      NOT elevatorReadyForAutomaticCycle OR
      elevatorFault THEN

    sheetStackDischargeFaultCode := 5;

ELSIF NOT synchronizedConveyorsRunning THEN

    sheetStackDischargeFaultCode := 6;

END_IF;


//==============================================================
// 6) Optional reset of current sequence fault display
//==============================================================
// EN: Reset clears the current sequence fault flag,
//     but does not erase last cycle diagnostic codes.
IF resetCmd AND (sheetStackDischargeControlState = 0) THEN

    sheetStackDischargeFault := FALSE;
    sheetStackDischargeFaultCode := 0;

END_IF;


//==============================================================
// 7) Arm discharge sequence from packageCompleteCmd
//==============================================================
// EN: packageCompleteCmd is ignored if the elevator is not in automatic,
//     the stacker is not running or a relevant drive/safety fault is active.
// PT: packageCompleteCmd é ignorado se o elevador não estiver em automático,
//     o stacker não estiver rodando ou houver falha relevante de drive/segurança.
IF rPackageCompleteDischarge AND
   elevatorAutoCmd AND
   synchronizedConveyorsRunning AND
   NOT sheetStackDischargeFaultCondition AND
   NOT sheetStackDischargeFault AND
   NOT sheetStackDischargeActive AND
   NOT sheetStackDischargePending THEN

    sheetStackDischargePending := TRUE;

    // EN: Clear current-cycle flags when a new cycle is accepted.
    sheetStackDischargeFault := FALSE;
    sheetStackDischargeFaultCode := 0;

    sheetStackDischargeCycleHasManualSkip := FALSE;
    sheetStackDischargeCycleHasTimeout := FALSE;

END_IF;


//==============================================================
// 8) Immediate abort condition
//==============================================================
// EN: Faults before discharge positioning cancel the request. Faults after
//     positioning starts hold safe targets until operator acknowledgement.
// PT: Falhas antes do posicionamento cancelam o pedido. Após o início,
//     mantêm os alvos seguros até o reconhecimento do operador.
abortCycle :=
    (
        sheetStackDischargeActive OR
        sheetStackDischargePending OR
        (sheetStackDischargeControlState <> 0)
    )
    AND
    (
        sheetStackDischargeFaultCondition OR
        NOT synchronizedConveyorsRunning
    );


IF abortCycle THEN

    sheetStackDischargeConveyorRunRequest := FALSE;
    sheetStackDischargePending := FALSE;

    tonSheetStackDischarge(IN := FALSE);
    tonSheetStackDischargeStepTimeout(IN := FALSE);
    tonSheetStackDischargePlatformClearTimeout(IN := FALSE);

    sheetStackDischargeFault := TRUE;

    sheetStackDischargeLastCycleOk := FALSE;
    sheetStackDischargeLastResultCode := 4;
    sheetStackDischargeLastFaultCode := sheetStackDischargeFaultCode;

    // EN: Do not clear backstopManualInterventionActive here.
    //     If the cycle aborted before return, keeping the memory is safer
    //     for the next cycle.

    IF sheetStackDischargeControlState <= 5 THEN

        // EN: No discharge movement has started yet.
        // PT: Nenhum movimento de descarte foi iniciado.
        sheetStackDischargeActive := FALSE;

        backstopTargetOverrideActive := FALSE;
        elevatorTargetOverrideActive := FALSE;

        elevatorPlatformClearDetected := FALSE;
        elevatorStackPresentAtDischargeStart := FALSE;

        sheetStackDischargeLastFaultStepCode :=
            sheetStackDischargeControlState;

        sheetStackDischargeState := 'ABORTED';
        sheetStackDischargeStateCode := 90;
        sheetStackDischargeControlState := 0;

    ELSE

        // EN: Preserve the original failed step while the external
        //     fault condition remains active in FAULT_HOLD.
        // PT: Preserva o passo original da falha enquanto a condição
        //     externa permanecer ativa no FAULT_HOLD.
        IF sheetStackDischargeControlState <> 90 THEN
            sheetStackDischargeLastFaultStepCode :=
                sheetStackDischargeControlState;
        END_IF;

        sheetStackDischargeActive := TRUE;
        sheetStackDischargeState := 'FAULT_HOLD';
        sheetStackDischargeStateCode := 90;

        IF sheetStackDischargeLastFaultStepCode < 40 THEN

            backstopTargetOverrideActive := TRUE;
            backstopTargetOverridePositionMm :=
                backstopDischargeOpenTargetMm;

            elevatorTargetOverrideActive := TRUE;
            elevatorTargetOverridePositionMm :=
                machineConfig.elevatorMinPositionMm;

        ELSE

            backstopTargetOverrideActive := TRUE;
            backstopTargetOverridePositionMm :=
                backstopProgrammedDischargeTargetMm;

            elevatorTargetOverrideActive := TRUE;
            elevatorTargetOverridePositionMm :=
                machineConfig.elevatorMaxPositionMm;

        END_IF;

        sheetStackDischargeControlState := 90;

    END_IF


ELSE

    //==============================================================
    // 9) Sheet stack discharge state machine
    //==============================================================
    CASE sheetStackDischargeControlState OF

        0: // IDLE
            sheetStackDischargeState := 'IDLE';
            sheetStackDischargeStateCode := 0;

            sheetStackDischargeActive := FALSE;

            sheetStackDischargeConveyorRunRequest := FALSE;

            backstopTargetOverrideActive := FALSE;
            elevatorTargetOverrideActive := FALSE;

            tonSheetStackDischarge(IN := FALSE);
            tonSheetStackDischargeStepTimeout(IN := FALSE);
            tonSheetStackDischargePlatformClearTimeout(IN := FALSE);
            elevatorPlatformClearDetected := FALSE;
            elevatorStackPresentAtDischargeStart := FALSE;

            IF sheetStackDischargePending THEN

                tonSheetStackDischarge(IN := FALSE);
                tonSheetStackDischargeStepTimeout(IN := FALSE);

                sheetStackDischargeControlState := 5;

            END_IF


        5: // WAIT_SEPARATION
            sheetStackDischargeState := 'WAIT_SEPARATION';
            sheetStackDischargeStateCode := 5;

            sheetStackDischargeActive := FALSE;

            sheetStackDischargeConveyorRunRequest := FALSE;

            backstopTargetOverrideActive := FALSE;
            elevatorTargetOverrideActive := FALSE;

            tonSheetStackDischarge(IN := FALSE);

            // EN: Wait for conveyor speed control to finish sheet stack separation.
            tonSheetStackDischargeStepTimeout(
                IN := TRUE,
                PT := machineConfig.sheetStackDischargeWaitSeparationTimeout
            );

            // EN: Complex stacker discharge starts only after conveyor 4
            //     completes the package separation sequence.
            // PT: O descarte do stacker complexo inicia somente depois que
            //     a esteira 4 concluir a sequência de separação do pacote.
            IF sheetStackSeparationFinished AND
               sheetConveyor4SeparationFinished THEN

                tonSheetStackDischargeStepTimeout(IN := FALSE);

                sheetStackDischargeControlState := 10;


            ELSIF tonSheetStackDischargeStepTimeout.Q THEN

                // EN: Separation did not finish. Do not discharge.
                tonSheetStackDischargeStepTimeout(IN := FALSE);

                sheetStackDischargePending := FALSE;
                sheetStackDischargeActive := FALSE;

                sheetStackDischargeFault := TRUE;
                sheetStackDischargeFaultCode := 10;

                sheetStackDischargeLastCycleOk := FALSE;
                sheetStackDischargeLastResultCode := 3;
                sheetStackDischargeLastFaultStepCode := 5;
                sheetStackDischargeLastFaultCode := 10;

                sheetStackDischargeControlState := 0;

            END_IF


        10: // START_DISCHARGE_POSITIONING
            sheetStackDischargeState := 'START_POSITIONING';
            sheetStackDischargeStateCode := 10;

            sheetStackDischargePending := FALSE;
            sheetStackDischargeActive := TRUE;
            sheetStackDischargeStarted := TRUE;

            elevatorPlatformClearDetected := FALSE;
            tonSheetStackDischargePlatformClearTimeout(IN := FALSE);
            elevatorStackPresentAtDischargeStart :=
                elevatorStackPresentSensor;

            tonSheetStackDischarge(IN := FALSE);
            tonSheetStackDischargeStepTimeout(IN := FALSE);

            //======================================================
            // EN: Latch programmed backstop target for this cycle.
            //     This is the normal position based on sheet length.
            //======================================================
            backstopProgrammedDischargeTargetMm :=
                LIMIT(
                    machineConfig.backstopMinPositionMm,
                    MAX(0.0, sheetLengthMm) +
                        machineConfig.backstopSheetLengthOffsetMm,
                    machineConfig.backstopMaxPositionMm
                );

            //======================================================
            // EN: Define safe opening base position.
            //
            // If the operator manually moved the backstop before the
            // automatic cycle, use the greater value between:
            // - programmed position
            // - last manual intervention position
            //
            // This prevents the automatic opening override from closing
            // the backstop onto the material.
            //
            // If there was no manual intervention, use only the programmed
            // position as the base.
            //======================================================
            IF backstopManualInterventionActive THEN

                backstopDischargeOpenBasePositionMm :=
                    MAX(
                        backstopProgrammedDischargeTargetMm,
                        backstopManualInterventionPositionMm
                    );

            ELSE

                backstopDischargeOpenBasePositionMm :=
                    backstopProgrammedDischargeTargetMm;

            END_IF;

            //======================================================
            // EN: Latch safe discharge open target.
            //     Offset is applied after selecting the safe base.
            //======================================================
            backstopDischargeOpenTargetMm :=
                LIMIT(
                    machineConfig.backstopMinPositionMm,
                    backstopDischargeOpenBasePositionMm +
                        machineConfig.backstopDischargeOpenOffsetMm,
                    machineConfig.backstopMaxPositionMm
                );

            // EN: Request safe backstop opening.
            //     Backstop control accepts it only in auto.
            backstopTargetOverrideActive := TRUE;
            backstopTargetOverridePositionMm := backstopDischargeOpenTargetMm;

            // EN: Request the elevator lower discharge position.
            // PT: Solicita a posição inferior de descarte do elevador.
            elevatorTargetOverrideActive := TRUE;
            elevatorTargetOverridePositionMm :=
                machineConfig.elevatorMinPositionMm;

            sheetStackDischargeControlState := 20;


        20: // WAIT_DISCHARGE_POSITION
            sheetStackDischargeState := 'WAIT_DISCHARGE_POS';
            sheetStackDischargeStateCode := 20;

            sheetStackDischargeActive := TRUE;

            // EN: Keep safe latched backstop discharge target active.
            backstopTargetOverrideActive := TRUE;
            backstopTargetOverridePositionMm := backstopDischargeOpenTargetMm;

            // EN: Keep the lower discharge target active and wait for feedback.
            // PT: Mantém o alvo inferior de descarte e aguarda o feedback.
            elevatorTargetOverrideActive := TRUE;
            elevatorTargetOverridePositionMm :=
                machineConfig.elevatorMinPositionMm;

            // EN: Discharge override controls the backstop automatically
            //     and blocks its manual commands during the cycle.
            // PT: O override de descarte controla o backstop automaticamente
            //     e bloqueia os comandos manuais durante o ciclo.
            backstopDischargeReady := backstopInPosition;

            IF backstopDischargeReady AND elevatorInPosition THEN

                tonSheetStackDischargeStepTimeout(IN := FALSE);
                sheetStackDischargeControlState := 30;

            ELSE

                tonSheetStackDischargeStepTimeout(
                    IN := TRUE,
                    PT := machineConfig.sheetStackDischargePositioningTimeout
                );

                IF tonSheetStackDischargeStepTimeout.Q THEN

